FUNCTION BOOLS_TO_DWORD
  (* Standard: 61499-1 *)
  (* Version 1.0, 2024-02-22, franz *)
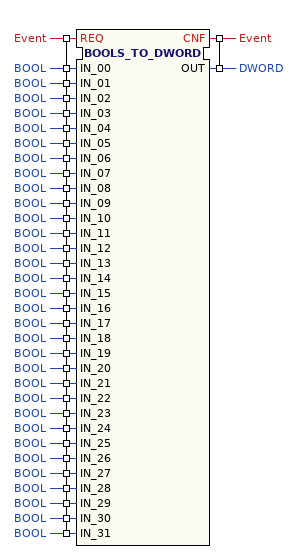
  EVENT_INPUT
    REQ WITH IN_00, IN_01, IN_02, IN_03, IN_04, IN_05, IN_06, IN_07, IN_08, IN_09, IN_10, IN_11, IN_12, IN_13, IN_14, IN_15, IN_16, IN_17, IN_18, IN_19, IN_20, IN_21, IN_22, IN_23, IN_24, IN_25, IN_26, IN_27, IN_28, IN_29, IN_30, IN_31; (* Normal Execution Request *)
  END_EVENT
  EVENT_OUTPUT
    CNF WITH OUT; (* Execution Confirmation *)
  END_EVENT
  VAR_INPUT
    IN_00 : BOOL; (* BIT 00 *)
    IN_01 : BOOL; (* BIT 01 *)
    IN_02 : BOOL; (* BIT 02 *)
    IN_03 : BOOL; (* BIT 03 *)
    IN_04 : BOOL; (* BIT 04 *)
    IN_05 : BOOL; (* BIT 05 *)
    IN_06 : BOOL; (* BIT 06 *)
    IN_07 : BOOL; (* BIT 07 *)
    IN_08 : BOOL; (* BIT 08 *)
    IN_09 : BOOL; (* BIT 09 *)
    IN_10 : BOOL; (* BIT 10 *)
    IN_11 : BOOL; (* BIT 11 *)
    IN_12 : BOOL; (* BIT 12 *)
    IN_13 : BOOL; (* BIT 13 *)
    IN_14 : BOOL; (* BIT 14 *)
    IN_15 : BOOL; (* BIT 15 *)
    IN_16 : BOOL; (* BIT 16 *)
    IN_17 : BOOL; (* BIT 17 *)
    IN_18 : BOOL; (* BIT 18 *)
    IN_19 : BOOL; (* BIT 19 *)
    IN_20 : BOOL; (* BIT 20 *)
    IN_21 : BOOL; (* BIT 21 *)
    IN_22 : BOOL; (* BIT 22 *)
    IN_23 : BOOL; (* BIT 23 *)
    IN_24 : BOOL; (* BIT 24 *)
    IN_25 : BOOL; (* BIT 25 *)
    IN_26 : BOOL; (* BIT 26 *)
    IN_27 : BOOL; (* BIT 27 *)
    IN_28 : BOOL; (* BIT 28 *)
    IN_29 : BOOL; (* BIT 29 *)
    IN_30 : BOOL; (* BIT 30 *)
    IN_31 : BOOL; (* BIT 31 *)
  END_VAR
  VAR_OUTPUT
    OUT : DWORD; (* DWORD Output *)
  END_VAR
  BODY IN ST:
FUNCTION BOOLS_TO_DWORD

VAR_INPUT
	IN_00 : BOOL;    // BIT 00
	IN_01 : BOOL;    // BIT 01
	IN_02 : BOOL;    // BIT 02
	IN_03 : BOOL;    // BIT 03
	IN_04 : BOOL;    // BIT 04
	IN_05 : BOOL;    // BIT 05
	IN_06 : BOOL;    // BIT 06
	IN_07 : BOOL;    // BIT 07
	IN_08 : BOOL;    // BIT 08
	IN_09 : BOOL;    // BIT 09
	IN_10 : BOOL;    // BIT 10
	IN_11 : BOOL;    // BIT 11
	IN_12 : BOOL;    // BIT 12
	IN_13 : BOOL;    // BIT 13
	IN_14 : BOOL;    // BIT 14
	IN_15 : BOOL;    // BIT 15
	IN_16 : BOOL;    // BIT 16
	IN_17 : BOOL;    // BIT 17
	IN_18 : BOOL;    // BIT 18
	IN_19 : BOOL;    // BIT 19
	IN_20 : BOOL;    // BIT 20
	IN_21 : BOOL;    // BIT 21
	IN_22 : BOOL;    // BIT 22
	IN_23 : BOOL;    // BIT 23
	IN_24 : BOOL;    // BIT 24
	IN_25 : BOOL;    // BIT 25
	IN_26 : BOOL;    // BIT 26
	IN_27 : BOOL;    // BIT 27
	IN_28 : BOOL;    // BIT 28
	IN_29 : BOOL;    // BIT 29
	IN_30 : BOOL;    // BIT 30
	IN_31 : BOOL;    // BIT 31
END_VAR

VAR_OUTPUT
	OUT : DWORD;    // DWORD Output
END_VAR

(* this Function combines the 32 BOOLS to a dword *)
OUT.0 := IN_00;
OUT.1 := IN_01;
OUT.2 := IN_02;
OUT.3 := IN_03;
OUT.4 := IN_04;
OUT.5 := IN_05;
OUT.6 := IN_06;
OUT.7 := IN_07;
OUT.8 := IN_08;
OUT.9 := IN_09;
OUT.10 := IN_10;
OUT.11 := IN_11;
OUT.12 := IN_12;
OUT.13 := IN_13;
OUT.14 := IN_14;
OUT.15 := IN_15;
OUT.16 := IN_16;
OUT.17 := IN_17;
OUT.18 := IN_18;
OUT.19 := IN_19;
OUT.20 := IN_20;
OUT.21 := IN_21;
OUT.22 := IN_22;
OUT.23 := IN_23;
OUT.24 := IN_24;
OUT.25 := IN_25;
OUT.26 := IN_26;
OUT.27 := IN_27;
OUT.28 := IN_28;
OUT.29 := IN_29;
OUT.30 := IN_30;
OUT.31 := IN_31;
END_FUNCTION
  END_BODY
END_FUNCTION
